FUNCTION_BLOCK MOD_OwnerLatch (* Local channel IDs of the occupation owner and its refresh query; types and forwards the received occupation owner *)
  (* Standard: 61499-2 *)
  (* Version 0.1, 2026-09-28, Project contributors, AAU Smart Production Lab *)
  PACKAGE modlib;
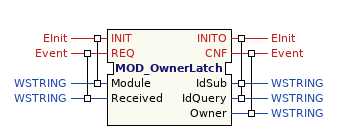
  EVENT_INPUT
    INIT : EInit WITH Module;
    REQ WITH Received;
  END_EVENT
  EVENT_OUTPUT
    INITO : EInit WITH IdSub, IdQuery;
    CNF WITH Owner;
  END_EVENT
  VAR_INPUT
    Module : WSTRING;
    Received : WSTRING;
  END_VAR
  VAR_OUTPUT
    IdSub : WSTRING;
    IdQuery : WSTRING;
    Owner : WSTRING;
  END_VAR
  EC_STATES
    INIT : INIT -> INITO;
    REQ : REQ -> CNF;
  END_STATES
  ALGORITHM INIT IN ST:
IdSub := CONCAT(CONCAT("loc[", Module), "/owner]");
IdQuery := CONCAT(CONCAT("loc[", Module), "/owner/query]");
  END_ALGORITHM
  ALGORITHM REQ IN ST:
Owner := Received;
  END_ALGORITHM
END_FUNCTION_BLOCK
